Yaskawa INFORM job: AAA.JBI

/JOB
//NAME AAA
//POS
///NPOS 3,0,0,0,0,0
///TOOL 9
///POSTYPE PULSE
///PULSE
C00000=-49828,124434,86505,3567,-56182,-4172
C00001=-48224,115593,74582,4243,-53470,-4916
C00002=-46571,108481,65128,4949,-51405,-5685
//INST
///DATE 2023/02/13 12:54
///ATTR SC,RW
///GROUP1 RB1
NOP
MOVJ C00000 VJ=1.0
MOVL C00001 V=5.0
MOVL C00002 V=5.0
END
